// TIA Portal V17 export
// export: Created 2022-07-20T06:59:46.5671773Z, ExportSetting WithDefaults, DisplayName Totally Integrated Automation Portal, DisplayVersion V17, DisplayName TIA Portal Openness, DisplayVersion V17, DisplayName TIA Portal Version Control Interface, DisplayVersion V17, DisplayName SINAMICS Startdrive Advanced, DisplayVersion V17, DisplayName SINAMICS Startdrive G130, G150, S120, S150, SINAMICS MV, S210, DisplayVersion V17, DisplayName SINAMICS Startdrive G110M, G120, G120C, G120D, G120P, G115D, DisplayVersion V17, DisplayName STEP 7 Professional, DisplayVersion V17, DisplayName STEP 7 Safety, DisplayVersion V17, DisplayName WinCC Advanced, DisplayVersion V17
FUNCTION_BLOCK "FB10096_ShutterEdgeDetection"   // FB10096, LAD
TITLE = Manage sheet edge detection
{ S7_Optimized_Access := 'TRUE' }
VERSION : 0.1
// stored: AutoNumber false, IsIECCheckEnabled false, IsRetainMemResEnabled false, MemoryReserve 100, SetENOAutomatically false, UDAEnableTagReadback false
   VAR_INPUT
      Enable { ExternalAccessible := 'False'; ExternalVisible := 'False'; ExternalWritable := 'False'} : Bool;
      Reset { ExternalAccessible := 'False'; ExternalVisible := 'False'; ExternalWritable := 'False'} : Bool;
   END_VAR
   VAR_OUTPUT
      Error { ExternalAccessible := 'False'; ExternalVisible := 'False'; ExternalWritable := 'False'} : Bool;
      SensorDetected : Bool;
      SensorActivated : Bool;
      SensorPositionDetected : LReal;
      DifferenceMeasured : LReal;
   END_VAR
   VAR_IN_OUT
      Sensor : TO_MeasuringInput;
   END_VAR
   VAR
      R_TRIG_Sensor { S7_SetPoint := 'True'} : R_TRIG;
      statSensorPosition { S7_SetPoint := 'True'} : LReal;
      statSensorPositionOld : LReal;
      statErrorMC : Bool;
      statSensorRisingEdgePosition : LReal;
      instMC_MEASURINGINPUT { S7_SetPoint := 'True'} : MC_MEASURINGINPUT;
   END_VAR
BEGIN

REGION Network 1 (SCL): Comments
   //==========================================================================================
   // SIEMENS SAS      RC-FR DI FA APC
   //------------------------------------------------------------------------------------------
   // Restrictions:    TIA V16 and more
   // Requirements:    S7-1500 + MGI library
   // Functionality:   This function block get position value of sheet edge 
   //------------------------------------------------------------------------------------------
   // Change log table:
   // Version      Date        Expert in charge    Changes applied
   // 01.00.01     09.06.2020  RTO                 First released version
   //==========================================================================================
END_REGION

REGION Network 2 (SCL): First Scan
   IF "FirstScan" THEN

       // Output
       #Error := FALSE;


       // Static
       #statSensorPosition := 0.0;
       #statSensorPositionOld := 0.0;
       #statErrorMC := FALSE;

   END_IF;
END_REGION

REGION Network 3 (SCL): Edge Signal Management
   REGION EDGE SIGNALS
       #R_TRIG_Sensor(CLK := #Sensor.InputState);
   END_REGION
END_REGION

REGION Network 4: Manage sensor acquisition
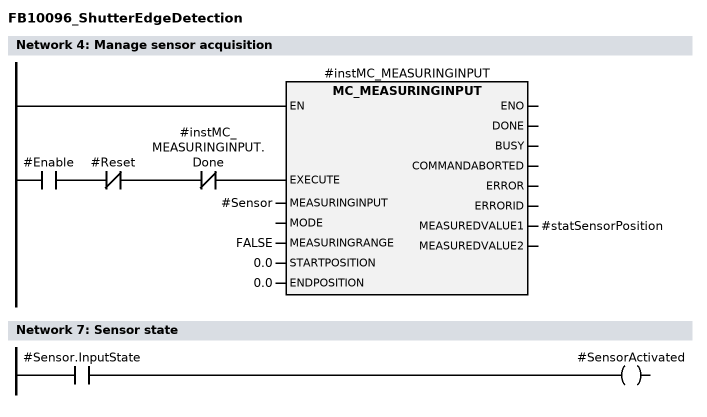
   RUNG wire#powerrail
      #instMC_MEASURINGINPUT.MC_MEASURINGINPUT(Execute := wire#w1, MeasuringInput := #Sensor, Mode :=, MeasuringRange := FALSE, StartPosition := 0.0, EndPosition := 0.0, Done =>, Busy =>, CommandAborted =>, Error =>, ErrorId =>, MeasuredValue1 => #statSensorPosition, MeasuredValue2 =>)
   END_RUNG
   RUNG wire#powerrail
      Contact( #Enable )
      I_Contact( #Reset )
      I_Contact( #instMC_MEASURINGINPUT.Done )
   END_RUNG wire#w1
   // the same network as SCL:
   #instMC_MEASURINGINPUT(Execute := #Enable AND NOT #Reset AND NOT #instMC_MEASURINGINPUT.Done,   // MC_MEASURINGINPUT
                          MeasuringInput := #Sensor,
                          MeasuringRange := FALSE,
                          StartPosition := 0.0,
                          EndPosition := 0.0,
                          MeasuredValue1 => #statSensorPosition);
END_REGION

REGION Network 5 (SCL): Manage sheet detection and position of synchronism
   IF #instMC_MEASURINGINPUT.Done THEN
       #SensorDetected := TRUE;
       #DifferenceMeasured := #statSensorPosition - #statSensorPositionOld;
       #SensorPositionDetected := #statSensorPosition;
       #statSensorPositionOld := #SensorPositionDetected;
       #statSensorRisingEdgePosition := #instMC_MEASURINGINPUT.MeasuredValue2;
   END_IF;

   IF #instMC_MEASURINGINPUT.Busy THEN
       #SensorDetected := FALSE;
   END_IF;

   IF #Reset THEN
       #SensorDetected := FALSE;
   END_IF;
END_REGION

REGION Network 6 (SCL): Manage error
   IF #statErrorMC THEN
       #Error := TRUE;
   ELSIF #Reset THEN
       #Error := FALSE;
   END_IF;
END_REGION

REGION Network 7: Sensor state
   RUNG wire#powerrail
      Contact( #Sensor.InputState )
      Coil( #SensorActivated )
   END_RUNG
   // the same network as SCL:
   #SensorActivated := #Sensor.InputState;
END_REGION
END_FUNCTION_BLOCK
